(* IEC 61131-3 sources: RL_MAR/experiments/comparison/llm4plc/results/gpt-4o-mini_20260506_100619/20260506_101558, 3 files *)

(* ---- generated_code_iteration_0.st ---- *)
ructured-text
FUNCTION_BLOCK HomeBrewingSystem
VAR_INPUT
    TemperatureSensor : REAL; (* Input for temperature measurement *)
    WaterFlowSensor : REAL; (* Input for water flow measurement *)
    BrewingStartTime : TIME; (* Input for brewing start time *)
    BrewingDuration : TIME; (* Input for brewing duration *)
END_VAR
VAR_OUTPUT
    HeatingElement : BOOL; (* Output for heating element *)
    AgitationMotor : BOOL; (* Output for agitation motor *)
    HopsDispenser : BOOL; (* Output for hops dispenser *)
    FermentationTank : BOOL; (* Output for fermentation tank *)
END_VAR
VAR
    state : INT; (* The state variable *)
    prevState : INT; (* The previous state variable *)
    brewingDurationInHours : INT; (* The brewing duration in hours *)
    temperature : REAL; (* The temperature variable *)
    waterFlow : REAL; (* The water flow variable *)
END_VAR

(* Initialize variables *)
state := 0;
prevState := 0;

(* Calculate brewing duration in hours *)
brewingDurationInHours := TO_INT(BrewingDuration / T#1h);

(* Control Logic *)
CASE state OF
    0: (* STATE 0: INITIALIZE *)
        HeatingElement := FALSE;
        AgitationMotor := FALSE;
        HopsDispenser := FALSE;
        FermentationTank := FALSE;
        state := 1; (* Transition to STATE 1 *)

    1: (* STATE 1: HEATING CONTROL *)
        IF TemperatureSensor < 65.0 THEN
            HeatingElement := TRUE;
        ELSE
            HeatingElement := FALSE;
        END_IF;
        state := 1; (* Remain in STATE 1 *)

    2: (* STATE 2: AGITATION CONTROL *)
        IF WaterFlowSensor > 0.5 THEN
            AgitationMotor := TRUE;
        ELSE
            AgitationMotor := FALSE;
        END_IF;
        state := 2; (* Remain in STATE 2 *)

    3: (* STATE 3: HOPS DISPENSING CONTROL *)
        IF brewingDurationInHours >= 5 THEN
            HopsDispenser := TRUE;
        ELSE
            HopsDispenser := FALSE;
        END_IF;
        state := 3; (* Remain in STATE 3 *)

    4: (* STATE 4: FERMENTATION CONTROL *)
        IF brewingDurationInHours >= 48 THEN
            FermentationTank := TRUE;
        ELSE
            FermentationTank := FALSE;
        END_IF;
        state := 4; (* Remain in STATE 4 *)

END_CASE;

END_FUNCTION_BLOCK

(* ---- generated_code_iteration_1.st ---- *)
START_REASON
The errors in the original Structured Text (ST) code occurred because the variable `BrewingDuration` was declared as a `TIME` type, but the code attempted to perform arithmetic operations on it, specifically dividing it by `T#1h`. This operation is not valid for the `TIME` type in Structured Text, leading to a type conversion error. To resolve this, the `BrewingDuration` should be converted to an appropriate type that allows for arithmetic operations, such as `UDINT`, which can represent the duration in milliseconds or seconds. Additionally, the variable section should be properly closed with `END_VAR` instead of `END_VAR_OUTPUT` or `END_VAR_INPUT`.
END_REASON

START_ST
FUNCTION_BLOCK HomeBrewingSystem
VAR_INPUT
    TemperatureSensor : REAL; (* Input for temperature measurement *)
    WaterFlowSensor : REAL; (* Input for water flow measurement *)
    BrewingStartTime : TIME; (* Input for brewing start time *)
    BrewingDuration : TIME; (* Input for brewing duration *)
END_VAR
VAR_OUTPUT
    HeatingElement : BOOL; (* Output for heating element *)
    AgitationMotor : BOOL; (* Output for agitation motor *)
    HopsDispenser : BOOL; (* Output for hops dispenser *)
    FermentationTank : BOOL; (* Output for fermentation tank *)
END_VAR
VAR
    state : INT; (* The state variable *)
    prevState : INT; (* The previous state variable *)
    brewingDurationInHours : INT; (* The brewing duration in hours *)
    temperature : REAL; (* The temperature variable *)
    waterFlow : REAL; (* The water flow variable *)
END_VAR

(* Initialize variables *)
state := 0;
prevState := 0;

(* Calculate brewing duration in hours *)
brewingDurationInHours := TO_INT(TO_UDINT(BrewingDuration) / T#1h);

(* Control Logic *)
CASE state OF
    0: (* STATE 0: INITIALIZE *)
        HeatingElement := FALSE;
        AgitationMotor := FALSE;
        HopsDispenser := FALSE;
        FermentationTank := FALSE;
        state := 1; (* Transition to STATE 1 *)

    1: (* STATE 1: HEATING CONTROL *)
        IF TemperatureSensor < 65.0 THEN
            HeatingElement := TRUE;
        ELSE
            HeatingElement := FALSE;
        END_IF;
        state := 1; (* Remain in STATE 1 *)

    2: (* STATE 2: AGITATION CONTROL *)
        IF WaterFlowSensor > 0.5 THEN
            AgitationMotor := TRUE;
        ELSE
            AgitationMotor := FALSE;
        END_IF;
        state := 2; (* Remain in STATE 2 *)

    3: (* STATE 3: HOPS DISPENSING CONTROL *)
        IF brewingDurationInHours >= 5 THEN
            HopsDispenser := TRUE;
        ELSE
            HopsDispenser := FALSE;
        END_IF;
        state := 3; (* Remain in STATE 3 *)

    4: (* STATE 4: FERMENTATION CONTROL *)
        IF brewingDurationInHours >= 48 THEN
            FermentationTank := TRUE;
        ELSE
            FermentationTank := FALSE;
        END_IF;
        state := 4; (* Remain in STATE 4 *)

END_CASE;

END_FUNCTION_BLOCK
END_ST

(* ---- generated_code_iteration_2.st ---- *)
START_REASON
The errors in the original Structured Text (ST) code occurred because the variable `BrewingDuration` was declared as a `TIME` type, but the code attempted to perform arithmetic operations on it, specifically dividing it by `T#1h`. This operation is not valid for the `TIME` type in Structured Text, leading to a type conversion error. To resolve this, the `BrewingDuration` should be converted to an appropriate type that allows for arithmetic operations, such as `UDINT`, which can represent the duration in milliseconds or seconds. Additionally, the variable section should be properly closed with `END_VAR` instead of `END_VAR_OUTPUT` or `END_VAR_INPUT`. In this corrected code, I will change the `BrewingDuration` from `TIME` to `UDINT` to allow for arithmetic operations.
END_REASON

START_ST
FUNCTION_BLOCK HomeBrewingSystem
VAR_INPUT
    TemperatureSensor : REAL; (* Input for temperature measurement *)
    WaterFlowSensor : REAL; (* Input for water flow measurement *)
    BrewingStartTime : TIME; (* Input for brewing start time *)
    BrewingDuration : UDINT; (* Input for brewing duration in milliseconds *)
END_VAR
VAR_OUTPUT
    HeatingElement : BOOL; (* Output for heating element *)
    AgitationMotor : BOOL; (* Output for agitation motor *)
    HopsDispenser : BOOL; (* Output for hops dispenser *)
    FermentationTank : BOOL; (* Output for fermentation tank *)
END_VAR
VAR
    state : INT; (* The state variable *)
    prevState : INT; (* The previous state variable *)
    brewingDurationInHours : INT; (* The brewing duration in hours *)
    temperature : REAL; (* The temperature variable *)
    waterFlow : REAL; (* The water flow variable *)
END_VAR

(* Initialize variables *)
state := 0;
prevState := 0;

(* Calculate brewing duration in hours *)
brewingDurationInHours := TO_INT(BrewingDuration / 3600000); (* Convert milliseconds to hours *)

(* Control Logic *)
CASE state OF
    0: (* STATE 0: INITIALIZE *)
        HeatingElement := FALSE;
        AgitationMotor := FALSE;
        HopsDispenser := FALSE;
        FermentationTank := FALSE;
        state := 1; (* Transition to STATE 1 *)

    1: (* STATE 1: HEATING CONTROL *)
        IF TemperatureSensor < 65.0 THEN
            HeatingElement := TRUE;
        ELSE
            HeatingElement := FALSE;
        END_IF;
        state := 1; (* Remain in STATE 1 *)

    2: (* STATE 2: AGITATION CONTROL *)
        IF WaterFlowSensor > 0.5 THEN
            AgitationMotor := TRUE;
        ELSE
            AgitationMotor := FALSE;
        END_IF;
        state := 2; (* Remain in STATE 2 *)

    3: (* STATE 3: HOPS DISPENSING CONTROL *)
        IF brewingDurationInHours >= 5 THEN
            HopsDispenser := TRUE;
        ELSE
            HopsDispenser := FALSE;
        END_IF;
        state := 3; (* Remain in STATE 3 *)

    4: (* STATE 4: FERMENTATION CONTROL *)
        IF brewingDurationInHours >= 48 THEN
            FermentationTank := TRUE;
        ELSE
            FermentationTank := FALSE;
        END_IF;
        state := 4; (* Remain in STATE 4 *)

END_CASE;

END_FUNCTION_BLOCK
END_ST
